TYPE E_StreamState :
(
	e_streamState_Pause := 0,
	e_streamState_Start		:=1,
	e_streamState_Select	:=2
);
END_TYPE

(* stored: Version 1.1.0.1, ProductVersion 3.1.4024.9
   DUT E_StreamState: Id {43a3f311-25f4-40f5-b8f2-2905f683bcc7} *)
